TYPE (* Telemetry connection config: wraps the MQTT_CONNECTION inputs *)
  (* Standard: 1131-3 *)
  (* Version 0.1, 6/21/2026, easensoy, WMG, single STRUCT input for Telemetry *)
  PACKAGE Main;
  TelemetryConfig : STRUCT
    QI : BOOL;
    ConnectionID : STRING[80];
    URL : STRING[255];
    ClientIdentifier : STRING[80];
    ValidateCert : USINT;
    CACert : STRING[255];
  END_STRUCT;
END_TYPE
